FUNCTION_BLOCK FB_RpcServer
VAR_INPUT
END_VAR
VAR_OUTPUT
END_VAR
VAR
END_VAR

{attribute 'TcRpcEnable'}
METHOD Greet : T_MaxString
VAR_INPUT
	sName : T_MaxString;
END_VAR
VAR_OUTPUT
	nLen : INT;
END_VAR
VAR_IN_OUT CONSTANT
	stLibVersion : ST_LibVersion;
END_VAR

Greet := CONCAT(CONCAT(CONCAT('Hello ', sName), '! LibVersion: '), stLibVersion.sVersion);

nLen := LEN(Greet);
END_METHOD

END_FUNCTION_BLOCK

(* stored: Version 1.1.0.1, ProductVersion 3.1.4024.12
   POU FB_RpcServer: Id {5415d0aa-1023-4e78-9aa7-017bf1acac92}, SpecialFunc None
   Method Greet: Id {61032f55-ad62-4559-be00-7ade16106678} *)
